DECL E6POS XCAux320={X -55.000,Y -4.290,Z 0.700,A 0.000,B 0.000,C -0.000}
DECL E6POS XCDes320={X 1.660,Y -16.330,Z 0.700,A 0.000,B 0.000,C -0.000}
;ENDDAT for Routine_0

ENDDAT
